FUNCTION_BLOCK FB_MotionRefSelector
VAR_INPUT
	Auto1Man0: BOOL;
	xCylRefGenm: LREAL;
	vCylRefGenm: LREAL;
	vCylJoyms: LREAL;
END_VAR
VAR_OUTPUT

END_VAR
VAR
	fbOpenLoopControl : FB_OpenLoopControl;
END_VAR

IF NOT(G_ControllerGreenCrane.eStatus = E_Status.Running) THEN 
	fbOpenLoopControl(bEnable := FALSE, fVelocityReference_ms := vCylJoyms, fMaxValveFlow_lmin := 19, fVelocityFeedForward => G_ControllerGreenCrane.fGain);
ELSIF NOT(Auto1Man0) THEN
    fbOpenLoopControl(bEnable := TRUE, fVelocityReference_ms := vCylJoyms, fMaxValveFlow_lmin := 19, fVelocityFeedForward => G_ControllerGreenCrane.fGain);
ELSE 
	fbOpenLoopControl(bEnable := FALSE, fVelocityReference_ms := vCylJoyms, fMaxValveFlow_lmin := 19, fVelocityFeedForward => G_ControllerGreenCrane.fGain); //This will be Auto
END_IF;

END_FUNCTION_BLOCK

(* stored: Version 1.1.0.1, ProductVersion 3.1.4024.12
   POU FB_MotionRefSelector: Id {8bb19fa7-05f7-4e62-b98b-816ae3bdfb6f}, SpecialFunc None *)
